// TIA Portal project "LinkedList_v000_000_008" (V16)
// task for 000.000.007: create LinkedList.Insert

(* hardware
DEVICE "S7-1200 station_1"  S7-1200 Station
   slot 0: "Rack_0"  S7-1200 Rack  Rack  V1.0
   slot 1: "PLC_1"  CPU 1212C DC/DC/DC  6ES7 212-1AE40-0XB0  V4.4
*)

// ===== PLC "PLC_1"  CPU 1212C DC/DC/DC =====

VAR_GLOBAL   // PLC tag table "Default tag table"
   "System_Byte" AT %MB1 : Byte;
   "FirstScan" AT %M1.0 : Bool;
   "DiagStatusUpdate" AT %M1.1 : Bool;
   "AlwaysTRUE" AT %M1.2 : Bool;
   "AlwaysFALSE" AT %M1.3 : Bool;
   "Clock_Byte" AT %MB0 : Byte;
   "Clock_10Hz" AT %M0.0 : Bool;
   "Clock_5Hz" AT %M0.1 : Bool;
   "Clock_2.5Hz" AT %M0.2 : Bool;
   "Clock_2Hz" AT %M0.3 : Bool;
   "Clock_1.25Hz" AT %M0.4 : Bool;
   "Clock_1Hz" AT %M0.5 : Bool;
   "Clock_0.625Hz" AT %M0.6 : Bool;
   "Clock_0.5Hz" AT %M0.7 : Bool;
END_VAR

VAR_GLOBAL CONSTANT   // PLC tag table "Default tag table"
   "NULL_TOKEN" : DInt := -1;
   "AVAILABLE_SLOT" : DInt := -1;
   "TAIL_ADDRESS" : DInt := -2;
   "NOT_FOUND_FLAG" : DInt := -1;
END_VAR

TYPE "LinkedList.Node.Payload.UDT"
   STRUCT
      id : Char;
      status : String;
   END_STRUCT;
END_TYPE

TYPE "LinkedList.Node.UDT"
   STRUCT
      payload : "LinkedList.Node.Payload.UDT";
      pointer : DInt := -1;
   END_STRUCT;
END_TYPE

TYPE "LinkedList.UDT"
   STRUCT
      head : DInt := -1;
      list : Array[0..4] of "LinkedList.Node.UDT";
   END_STRUCT;
END_TYPE

TYPE "Validate.LinkedList.FindPointer.UDT"
   STRUCT
      request : Bool;
      needle : DInt;
      not_found : DInt;
      index : DInt;
   END_STRUCT;
END_TYPE

TYPE "Validate.LinkedList.FindPayload.UDT"
   STRUCT
      request : Bool;
      needle : "LinkedList.Node.Payload.UDT";
      not_found : DInt;
      tail_address : DInt;
      index : DInt;
   END_STRUCT;
END_TYPE

TYPE "Validate.LinkedList.FindID.UDT"
   STRUCT
      request : Bool;
      needle : Char;
      not_found : DInt;
      tail_address : DInt;
      index : DInt;
   END_STRUCT;
END_TYPE

TYPE "Validate.LinkedList.FindStatus.UDT"
   STRUCT
      request : Bool;
      needle : String;
      not_found : DInt;
      tail_address : DInt;
      index : DInt;
   END_STRUCT;
END_TYPE

TYPE "Validate.LinkedList.AddHead.UDT"
   STRUCT
      request : Bool;
      available_slot : DInt := -1;
      payload : "LinkedList.Node.Payload.UDT";
      tail_address : DInt := -2;
      status : String;
   END_STRUCT;
END_TYPE

TYPE "Validate.LinkedList.RemoveHead.UDT"
   STRUCT
      request : Bool;
      status : String;
   END_STRUCT;
END_TYPE

TYPE "Validate.LinkedList.FindPrevious.UDT"
   STRUCT
      request : Bool;
      needle : "LinkedList.Node.Payload.UDT";
      not_found : DInt;
      tail_address : DInt;
      index : DInt;
   END_STRUCT;
END_TYPE

TYPE "Validate.LinkedList.RemoveNode.UDT"
   STRUCT
      request : Bool;
      payload : "LinkedList.Node.Payload.UDT";
      null_token : DInt := -1;
      tail_address : DInt := -2;
      status : String;
   END_STRUCT;
END_TYPE

TYPE "Validate.LinkedList.Append.UDT"
   STRUCT
      request : Bool;
      payload : "LinkedList.Node.Payload.UDT";
      available_slot : DInt := -1;
      tail_address : DInt := -2;
      status : String;
   END_STRUCT;
END_TYPE

TYPE "Validate.LinkedList.Insert.UDT"
   STRUCT
      request : Bool;
      payload : "LinkedList.Node.Payload.UDT";
      after : "LinkedList.Node.Payload.UDT";
      available_slot : DInt := -1;
      not_found : DInt := -1;
      tail_address : DInt := -2;
      status : String;
   END_STRUCT;
END_TYPE

TYPE "Validate.LinkedList.Clear.UDT"
   STRUCT
      request : Bool;
      available_slot : DInt := -1;
      tail_address : DInt := -2;
      status : String;
   END_STRUCT;
END_TYPE

TYPE "Validate.LinkedList.AddNode.UDT"
   STRUCT
      request : Bool;
      available_slot : DInt := -1;
      payload : "LinkedList.Node.Payload.UDT";
      tail_address : DInt := -2;
      status : String;
   END_STRUCT;
END_TYPE

DATA_BLOCK "LinkedList.IDB"   // DB1
{ S7_Optimized_Access := 'TRUE' }
AUTHOR : Machado
FAMILY : LinkedList
VERSION : 0.1
// stored: InstanceOfName LinkedList
"LinkedList"
BEGIN
END_DATA_BLOCK

DATA_BLOCK "ValidationSignals"   // DB2
{ S7_Optimized_Access := 'TRUE' }
VERSION : 0.1
   VAR
      FindPointer : "Validate.LinkedList.FindPointer.UDT";
      FindPayload : "Validate.LinkedList.FindPayload.UDT";
      FindID : "Validate.LinkedList.FindID.UDT";
      FindStatus : "Validate.LinkedList.FindStatus.UDT";
      AddHead : "Validate.LinkedList.AddHead.UDT";
      RemoveHead : "Validate.LinkedList.RemoveHead.UDT";
      FindPrevious : "Validate.LinkedList.FindPrevious.UDT";
      RemoveNode : "Validate.LinkedList.RemoveNode.UDT";
      AppendNode : "Validate.LinkedList.Append.UDT";
      InsertNode : "Validate.LinkedList.Insert.UDT";
      Clear : "Validate.LinkedList.Clear.UDT";
      AddNode : "Validate.LinkedList.AddNode.UDT";
   END_VAR
BEGIN
END_DATA_BLOCK

FUNCTION_BLOCK "LinkedList"   // FB1, SCL
TITLE = Linked List
{ S7_Optimized_Access := 'TRUE' }
AUTHOR : Machado
FAMILY : LinkedList
VERSION : 0.1
   VAR_INPUT
      request : DInt;
   END_VAR
   VAR
      list : "LinkedList.UDT";
      requests : "LinkedList.UDT";
   END_VAR
   VAR_TEMP
      test : DInt;
   END_VAR
BEGIN
   CASE #request OF
       0:  // Statement section case 1
           ;
       2..4:  // Statement section case 2 to 4
           ;
       ELSE  // Statement section ELSE
           ;
   END_CASE;
END_FUNCTION_BLOCK

FUNCTION "LinkedList.FindPointer" : DInt   // FC1, SCL
TITLE = Find Node by Pointer In Linked List
{ S7_Optimized_Access := 'TRUE' }
AUTHOR : Machado
FAMILY : LinkedList
VERSION : 0.1
// returns not_found when not found.
// otherwise returs index of parent array where node with needle value as pointer.
   VAR_INPUT
      needle : DInt;
      not_found : DInt;   // value returned to user if needle not found
   END_VAR
   VAR_IN_OUT
      haystack : "LinkedList.UDT";
   END_VAR
   VAR_TEMP
      i : DInt;
      size : DInt;
   END_VAR
BEGIN
   REGION "GET SIZE"
       #size := UDINT_TO_DINT("LinkedList.Node[].CountOfElements"(#haystack.list));
   END_REGION


   REGION "SEARCH"
       FOR #i := 0 TO #size - 1 DO
           // no match
           IF #haystack.list[#i]."pointer" <> #needle THEN
               CONTINUE;
           END_IF;
           // match
           #"LinkedList.FindPointer" := #i;
           RETURN;
       END_FOR;
   END_REGION


   REGION "NOT FOUND"
       #"LinkedList.FindPointer" := #not_found;
       RETURN;
   END_REGION
END_FUNCTION

FUNCTION "LinkedList.Node[].CountOfElements" : UDInt   // FC2, SCL
TITLE = Count Of Elements of an Array of Linked List Nodes
{ S7_Optimized_Access := 'TRUE' }
AUTHOR : Machado
FAMILY : LinkedList
VERSION : 0.1
   VAR_INPUT
      list : Variant;
   END_VAR
BEGIN
   #"LinkedList.Node[].CountOfElements" := CountOfElements(#list);
   RETURN;
END_FUNCTION

FUNCTION "LinkedList.FindPayload" : DInt   // FC3, SCL
TITLE = Finde Node Index By Payload
{ S7_Optimized_Access := 'TRUE' }
AUTHOR : Machado
FAMILY : LinkedList
VERSION : 0.1
   VAR_INPUT
      needle : "LinkedList.Node.Payload.UDT";
      not_found : DInt;
      tail_address : DInt;
   END_VAR
   VAR_IN_OUT
      haystack : "LinkedList.UDT";
   END_VAR
   VAR_TEMP
      size : DInt;
      this_node : "LinkedList.Node.UDT";
      next_node : "LinkedList.Node.UDT";
      nodes_visited : DInt;
   END_VAR
BEGIN
   REGION "GET SIZE"
       #size := UDINT_TO_DINT("LinkedList.Node[].CountOfElements"(#haystack.list));
   END_REGION


   REGION "PRE-CONDITIONS"
       IF NOT "DInt.InRange"(x := #haystack.head, max := #size - 1, min := 0) THEN
           #"LinkedList.FindPayload" := #not_found;
           RETURN;
       END_IF;
   END_REGION


   REGION "PRIME WHILE LOOP"
       #this_node := #haystack.list[#haystack.head];
       IF #this_node.payload = #needle THEN
           #"LinkedList.FindPayload" := #haystack.head;
           RETURN;
       END_IF;
       #nodes_visited := 1;
   END_REGION


   REGION "SEARCH"
       WHILE #this_node."pointer" <> #tail_address DO
           #next_node := #haystack.list[#this_node."pointer"];
           IF #next_node.payload = #needle THEN
               #"LinkedList.FindPayload" := #this_node."pointer";
               RETURN;
           END_IF;
           #nodes_visited += 1;
           IF #nodes_visited > #size THEN
               #"LinkedList.FindPayload" := #not_found;
               RETURN;
           END_IF;
           #this_node := #next_node;
       END_WHILE;
   END_REGION


   REGION "NOT FOUND"
       #"LinkedList.FindPayload" := #not_found;
       RETURN;
   END_REGION
END_FUNCTION

FUNCTION "DInt.InRange" : Bool   // FC4, SCL
TITLE = Value Is In Range
{ S7_Optimized_Access := 'TRUE' }
AUTHOR : Machado
FAMILY : DInt
VERSION : 0.1
   VAR_INPUT
      x : DInt;
      max : DInt;
      min : DInt;
   END_VAR
BEGIN
   #"DInt.InRange" := #min <= #x AND #x <= #max;
END_FUNCTION

FUNCTION "LinkedList.FindID" : DInt   // FC5, SCL
TITLE = Finde Node Index By Payload
{ S7_Optimized_Access := 'TRUE' }
AUTHOR : Machado
FAMILY : LinkedList
VERSION : 0.1
   VAR_INPUT
      needle : Char;
      not_found : DInt;
      tail_address : DInt;
   END_VAR
   VAR_IN_OUT
      haystack : "LinkedList.UDT";
   END_VAR
   VAR_TEMP
      size : DInt;
      this_node : "LinkedList.Node.UDT";
      next_node : "LinkedList.Node.UDT";
      nodes_visited : DInt;
   END_VAR
BEGIN
   REGION "GET SIZE"
       #size := UDINT_TO_DINT("LinkedList.Node[].CountOfElements"(#haystack.list));
   END_REGION


   REGION "PRE-CONDITIONS"
       IF NOT "DInt.InRange"(x := #haystack.head, max := #size - 1, min := 0) THEN
           #"LinkedList.FindID" := #not_found;
           RETURN;
       END_IF;
   END_REGION


   REGION "PRIME WHILE LOOP"
       #this_node := #haystack.list[#haystack.head];
       IF #this_node.payload.id = #needle THEN
           #"LinkedList.FindID" := #haystack.head;
           RETURN;
       END_IF;
       #nodes_visited := 1;
   END_REGION


   REGION "SEARCH"
       WHILE #this_node."pointer" <> #tail_address DO
           #next_node := #haystack.list[#this_node."pointer"];
           IF #next_node.payload.id = #needle THEN
               #"LinkedList.FindID" := #this_node."pointer";
               RETURN;
           END_IF;
           #nodes_visited += 1;
           IF #nodes_visited > #size THEN
               #"LinkedList.FindID" := #not_found;
               RETURN;
           END_IF;
           #this_node := #next_node;
       END_WHILE;
   END_REGION


   REGION "NOT FOUND"
       #"LinkedList.FindID" := #not_found;
       RETURN;
   END_REGION
END_FUNCTION

FUNCTION "LinkedList.FindStatus" : DInt   // FC6, SCL
TITLE = Finde Node Index By Payload
{ S7_Optimized_Access := 'TRUE' }
AUTHOR : Machado
FAMILY : LinkedList
VERSION : 0.1
   VAR_INPUT
      needle : String;
      not_found : DInt;
      tail_address : DInt;
   END_VAR
   VAR_IN_OUT
      haystack : "LinkedList.UDT";
   END_VAR
   VAR_TEMP
      size : DInt;
      this_node : "LinkedList.Node.UDT";
      next_node : "LinkedList.Node.UDT";
      nodes_visited : DInt;
   END_VAR
BEGIN
   REGION "GET SIZE"
       #size := UDINT_TO_DINT("LinkedList.Node[].CountOfElements"(#haystack.list));
   END_REGION


   REGION "PRE-CONDITIONS"
       IF NOT "DInt.InRange"(x := #haystack.head, max := #size - 1, min := 0) THEN
           #"LinkedList.FindStatus" := #not_found;
           RETURN;
       END_IF;
   END_REGION


   REGION "PRIME WHILE LOOP"
       #this_node := #haystack.list[#haystack.head];
       IF #this_node.payload.status = #needle THEN
           #"LinkedList.FindStatus" := #haystack.head;
           RETURN;
       END_IF;
       #nodes_visited := 1;
   END_REGION


   REGION "SEARCH"
       WHILE #this_node."pointer" <> #tail_address DO
           #next_node := #haystack.list[#this_node."pointer"];
           IF #next_node.payload.status = #needle THEN
               #"LinkedList.FindStatus" := #this_node."pointer";
               RETURN;
           END_IF;
           #nodes_visited += 1;
           IF #nodes_visited > #size THEN
               #"LinkedList.FindStatus" := #not_found;
               RETURN;
           END_IF;
           #this_node := #next_node;
       END_WHILE;
   END_REGION


   REGION "NOT FOUND"
       #"LinkedList.FindStatus" := #not_found;
       RETURN;
   END_REGION
END_FUNCTION

FUNCTION "LinkedList.AddHead" : String   // FC7, SCL
TITLE = Add a Head Node to a Linked List
{ S7_Optimized_Access := 'TRUE' }
AUTHOR : Machado
FAMILY : LinkedList
VERSION : 0.1
// Use this in your linked list. Instantiates LinkedList.CreateHead and LinkedList.ReplaceHead when appropriate.
   VAR_INPUT
      available_slot : DInt;
      payload : "LinkedList.Node.Payload.UDT";
      tail_address : DInt;
   END_VAR
   VAR_IN_OUT
      list : "LinkedList.UDT";
   END_VAR
   VAR_TEMP
      message : String;
   END_VAR
BEGIN
   REGION "NO HEAD"
       IF #list.head = -1 THEN
           #message := "LinkedList.CreateHead"(available_slot := #available_slot,
                                               payload := #payload,
                                               tail_address := #tail_address,
                                               list := #list);
           #"LinkedList.AddHead" := #message;
           RETURN;
       END_IF;
   END_REGION
   REGION "REPLACE HEAD"
       #message := "LinkedList.ReplaceHead"(available_slot := #available_slot,
                                            payload := #payload,
                                            tail_address := #tail_address,
                                            list := #list);
       #"LinkedList.AddHead" := #message;
       RETURN;
   END_REGION
END_FUNCTION

FUNCTION "LinkedList.CreateHead" : String   // FC8, SCL
TITLE = Create a New Head Node for a Linked List
{ S7_Optimized_Access := 'TRUE' }
AUTHOR : Machado
FAMILY : LinkedList
VERSION : 0.1
   VAR_INPUT
      available_slot : DInt;
      payload : "LinkedList.Node.Payload.UDT";
      tail_address : DInt;
   END_VAR
   VAR_IN_OUT
      list : "LinkedList.UDT";
   END_VAR
   VAR_TEMP
      first_available_slot : DInt;
      message : String;
   END_VAR
   VAR CONSTANT
      CREATED : String := 'head created';
      FULL : String := 'no space in array. head not created.';
      NOT_FOUND : DInt := -1;
   END_VAR
BEGIN
   REGION "GET FIRST AVAILABLE SLOT"
       #first_available_slot := "LinkedList.FindPointer"(needle := #available_slot,
                                                         not_found := #NOT_FOUND,
                                                         haystack := #list);
   END_REGION


   REGION "NO ROOM IN LIST"
       IF #first_available_slot = #NOT_FOUND THEN
           #"LinkedList.CreateHead" := #FULL;
           RETURN;
       END_IF;
   END_REGION


   REGION "CREATE HEAD"
       #message := "LinkedList.Clear"(available_slot := #available_slot,
                                      tail_address := #tail_address,
                                      list := #list);
       #list.head := #first_available_slot;
       #list.list[#first_available_slot].payload := #payload;
       #list.list[#first_available_slot]."pointer" := #tail_address;
       #"LinkedList.CreateHead" := #CREATED;
       RETURN;
   END_REGION
END_FUNCTION

FUNCTION "LinkedList.ReplaceHead" : String   // FC9, SCL
TITLE = Replace Linked List's Existing Head Node
{ S7_Optimized_Access := 'TRUE' }
AUTHOR : Machado
FAMILY : LinkedList
VERSION : 0.1
   VAR_INPUT
      available_slot : DInt;
      payload : "LinkedList.Node.Payload.UDT";
      tail_address : DInt;
   END_VAR
   VAR_IN_OUT
      list : "LinkedList.UDT";
   END_VAR
   VAR_TEMP
      first_available_slot : DInt;
   END_VAR
   VAR CONSTANT
      FULL : String := 'no space in array. new head not added.';
      ADDED : String := 'new head added';
      NOT_FOUND : DInt := -1;
   END_VAR
BEGIN
   REGION "GET FIRST AVAILABLE SLOT"
       #first_available_slot := "LinkedList.FindPointer"(needle := #available_slot,
                                                         not_found := #NOT_FOUND,
                                                         haystack := #list);
   END_REGION


   REGION "NO ROOM IN LIST"
       IF #first_available_slot = #NOT_FOUND THEN
           #"LinkedList.ReplaceHead" := #FULL;
           RETURN;
       END_IF;
   END_REGION


   REGION "CREATE HEAD"
       #list.list[#first_available_slot].payload := #payload;
       #list.list[#first_available_slot]."pointer" := #list.head;
       #list.head := #first_available_slot;
       #"LinkedList.ReplaceHead" := #ADDED;
       RETURN;
   END_REGION
END_FUNCTION

FUNCTION "LinkedList.DeleteNode" : "LinkedList.Node.UDT"   // FC10, SCL
TITLE = Delete a Node from a Linked List
{ S7_Optimized_Access := 'TRUE' }
AUTHOR : Machado
FAMILY : LinkedList
VERSION : 0.1
   VAR_INPUT
      null_token : DInt;
   END_VAR
   VAR_TEMP
      node : "LinkedList.Node.UDT";
   END_VAR
BEGIN
   #node."pointer" := #null_token;
   #"LinkedList.DeleteNode" := #node;
   RETURN;
END_FUNCTION

FUNCTION "LinkedList.RemoveHead" : String   // FC11, SCL
TITLE = Remove Head Node from a Linked List
{ S7_Optimized_Access := 'TRUE' }
AUTHOR : Machado
FAMILY : LinkedList
VERSION : 0.1
// no head: returns no head message
// has head: removes, returns removed head message
   VAR_INPUT
      null_token : DInt;
   END_VAR
   VAR_IN_OUT
      list : "LinkedList.UDT";
   END_VAR
   VAR_TEMP
      head_pointer : DInt;
   END_VAR
   VAR CONSTANT
      NO_HEAD : String := 'no head, no operation';
      HEAD_REMOVED : String := 'head removed';
      HEAD_INDEX_OUT_OF_BOUNDS : String := 'head index out of bounds. no operation.';
   END_VAR
BEGIN
   REGION "NO HEAD"
       IF #list.head < 0 THEN
           #"LinkedList.RemoveHead" := #NO_HEAD;
           RETURN;
       END_IF;
   END_REGION


   REGION "HEAD POINTER IS OUT OF BOUNDS"
       IF #list.head >= UDINT_TO_DINT("LinkedList.Node[].CountOfElements"(#list.list))THEN
           #"LinkedList.RemoveHead" := #HEAD_INDEX_OUT_OF_BOUNDS;
           RETURN;
       END_IF;
   END_REGION


   REGION "HAS HEAD"
       #head_pointer := #list.list[#list.head]."pointer";
       #list.list[#list.head] := "LinkedList.DeleteNode"(#null_token);
       #list.head := #head_pointer;
       #"LinkedList.RemoveHead" := #HEAD_REMOVED;
       RETURN;
   END_REGION
END_FUNCTION

FUNCTION "LinkedList.FindPrevious" : DInt   // FC12, SCL
TITLE = Finde Node Index By Payload
{ S7_Optimized_Access := 'TRUE' }
AUTHOR : Machado
FAMILY : LinkedList
VERSION : 0.1
   VAR_INPUT
      needle : "LinkedList.Node.Payload.UDT";
      not_found : DInt;
      tail_address : DInt;
   END_VAR
   VAR_IN_OUT
      haystack : "LinkedList.UDT";
   END_VAR
   VAR_TEMP
      size : DInt;
      this_node : "LinkedList.Node.UDT";
      this_node_index : DInt;
      next_node : "LinkedList.Node.UDT";
      nodes_visited : DInt;
   END_VAR
BEGIN
   REGION "GET SIZE"
       #size := UDINT_TO_DINT("LinkedList.Node[].CountOfElements"(#haystack.list));
   END_REGION


   REGION "PRE-CONDITIONS"
       IF NOT "DInt.InRange"(x := #haystack.head, max := #size - 1, min := 0) THEN
           #"LinkedList.FindPrevious" := #not_found;
           RETURN;
       END_IF;
   END_REGION


   REGION "PRIME WHILE LOOP"
       #this_node_index := #haystack.head;
       #this_node := #haystack.list[#haystack.head];
       IF #this_node.payload = #needle THEN
           #"LinkedList.FindPrevious" := #not_found;
           RETURN;
       END_IF;
       #nodes_visited := 1;
   END_REGION


   REGION "SEARCH"
       WHILE #this_node."pointer" <> #tail_address DO
           #next_node := #haystack.list[#this_node."pointer"];
           IF #next_node.payload = #needle THEN
               #"LinkedList.FindPrevious" := #this_node_index;
               RETURN;
           END_IF;
           #nodes_visited += 1;
           IF #nodes_visited >= #size THEN
               #"LinkedList.FindPrevious" := #not_found;
               RETURN;
           END_IF;
           #this_node_index := #this_node."pointer";
           #this_node := #next_node;
       END_WHILE;
   END_REGION


   REGION "NOT FOUND"
       #"LinkedList.FindPrevious" := #not_found;
       RETURN;
   END_REGION
END_FUNCTION

FUNCTION "LinkedList.RemoveNode" : String   // FC13, SCL
TITLE = Removes a Node From a Linked List
{ S7_Optimized_Access := 'TRUE' }
AUTHOR : Machado
FAMILY : LinkedList
VERSION : 0.1
   VAR_INPUT
      node_payload : "LinkedList.Node.Payload.UDT";
      null_token : DInt;
      tail_address : DInt;
   END_VAR
   VAR_IN_OUT
      list : "LinkedList.UDT";
   END_VAR
   VAR_TEMP
      previous_node_index : DInt;
      this_node_index : DInt;
      list_size : DInt;
   END_VAR
   VAR CONSTANT
      EMPTY_LIST : String := 'list empty. no operation.';
      NOT_FOUND : String := 'payload not found. no operation.';
      INVALID_INDEX : String := 'node found but at invalid array index. no operation.';
      SUCCESS : String := 'node removed from list.';
   END_VAR
BEGIN
   REGION "LIST IS EMPTY"
       IF #list.head < 0 THEN
           #"LinkedList.RemoveNode" := #EMPTY_LIST;
           RETURN;
       END_IF;
   END_REGION


   REGION "GET PREVIOUS NODE INDEX"
       #previous_node_index := "LinkedList.FindPrevious"(needle := #node_payload,
                                                         not_found := #null_token,
                                                         tail_address := #tail_address,
                                                         haystack := #list);
   END_REGION


   REGION "NODE NOT FOUND"
       IF #previous_node_index = #null_token THEN
           #"LinkedList.RemoveNode" := #NOT_FOUND;
           RETURN;
       END_IF;
   END_REGION


   REGION "GET THIS NODE INDEX"
       #this_node_index := #list.list[#previous_node_index]."pointer";
   END_REGION


   REGION "FOUND NODE INDEX INVALID"
       #list_size := UDINT_TO_DINT("LinkedList.Node[].CountOfElements"(#list.list));
       IF NOT "DInt.InRange"(x := #previous_node_index, max := #list_size - 1, min := 0) THEN
           #"LinkedList.RemoveNode" := #INVALID_INDEX;
           RETURN;
       END_IF;
       IF NOT "DInt.InRange"(x := #this_node_index, max := #list_size - 1, min := 0) THEN
           #"LinkedList.RemoveNode" := #INVALID_INDEX;
           RETURN;
       END_IF;
   END_REGION


   REGION "REMOVE"
       #list.list[#previous_node_index]."pointer" := #list.list[#this_node_index]."pointer";
       #list.list[#this_node_index] := "LinkedList.DeleteNode"(#null_token);
       #"LinkedList.RemoveNode" := #SUCCESS;
       RETURN;
   END_REGION
END_FUNCTION

FUNCTION "LinkedList.AppendNode" : String   // FC14, SCL
TITLE = Append New Node to End of Linked List
{ S7_Optimized_Access := 'TRUE' }
AUTHOR : Machado
FAMILY : LinkedList
VERSION : 0.1
   VAR_INPUT
      available_slot : DInt;
      payload : "LinkedList.Node.Payload.UDT";
      tail_address : DInt;
   END_VAR
   VAR_IN_OUT
      list : "LinkedList.UDT";
   END_VAR
   VAR_TEMP
      first_slot : DInt;
      size : DInt;
      tail : DInt;
   END_VAR
   VAR CONSTANT
      NOT_FOUND : DInt := -1;
      NO_AVAILABLE_SLOT : String := 'no available slot. no operation.';
      TAIL_NOT_FOUND : String := 'tail node not found. no operation.';
      TAIL_INDEX_NOT_IN_RANGE : String := 'tail index not in range. no operation';
      NODE_APPENDED : String := 'node appended';
   END_VAR
BEGIN
   REGION "GET FIRST SLOT"
       #first_slot := "LinkedList.FindPointer"(needle := #available_slot,
                                               not_found := #NOT_FOUND,
                                               haystack := #list);
   END_REGION


   REGION "NO SLOT AVAILABLE"
       IF #first_slot = #NOT_FOUND THEN
           #"LinkedList.AppendNode" := #NO_AVAILABLE_SLOT;
           RETURN;
       END_IF;
   END_REGION


   REGION "GET TAIL INDEX"
       #tail := "LinkedList.FindPointer"(needle := #tail_address,
                                         not_found := #NOT_FOUND,
                                         haystack := #list);
   END_REGION


   REGION "TAIL NOT FOUND"
       IF #tail = #NOT_FOUND THEN
           #"LinkedList.AppendNode" := #TAIL_NOT_FOUND;
           RETURN;
       END_IF;
   END_REGION


   REGION "TAIL INDEX NOT IN RANGE"
       #size := UDINT_TO_DINT("LinkedList.Node[].CountOfElements"(#list.list));
       IF NOT "DInt.InRange"(x := #tail, max := #size - 1, min := 0) THEN
           #"LinkedList.AppendNode" := #TAIL_INDEX_NOT_IN_RANGE;
           RETURN;
       END_IF;
   END_REGION


   REGION "APPEND"
       #list.list[#tail]."pointer" := #first_slot;
       #list.list[#first_slot].payload := #payload;
       #list.list[#first_slot]."pointer" := #tail_address;
       #"LinkedList.AppendNode" := #NODE_APPENDED;
       RETURN;
   END_REGION
END_FUNCTION

FUNCTION "LinkedList.InsertNode" : String   // FC15, SCL
TITLE = Insert a New Node into a Linked List
{ S7_Optimized_Access := 'TRUE' }
AUTHOR : Machado
FAMILY : LinkedList
VERSION : 0.1
   VAR_INPUT
      payload : "LinkedList.Node.Payload.UDT";
      after : "LinkedList.Node.Payload.UDT";
      available_slot : DInt;
      tail_address : DInt;
   END_VAR
   VAR_IN_OUT
      list : "LinkedList.UDT";
   END_VAR
   VAR_TEMP
      after_index : DInt;
      available_index : DInt;
      message : String;
      size : DInt;
   END_VAR
   VAR CONSTANT
      NOT_FOUND : DInt := -1;
      NO_AVAILABLE_SLOT : String := 'no available slot in parent array. no operation.';
      AFTER_NOT_FOUND : String := '"after" node not found. no operation.';
      NODE_INSERTED : String := 'node inserted.';
      AFTER_INDEX_INVALID : String := '"after" node index invalid. no operation.';
   END_VAR
BEGIN
   REGION "SLOT NOT AVAILABLE"
       #available_index := "LinkedList.FindPointer"(needle := #available_slot,
                                               not_found := #NOT_FOUND,
                                               haystack := #list);
       IF #available_index = #NOT_FOUND THEN
           #"LinkedList.InsertNode" := #NO_AVAILABLE_SLOT;
           RETURN;
       END_IF;
   END_REGION


   REGION "AFTER NODE NOT FOUND"
       #after_index := "LinkedList.FindPayload"(needle := #after,
                                                not_found := #NOT_FOUND,
                                                tail_address := #tail_address,
                                                haystack := #list);
       IF #after_index = #NOT_FOUND THEN
           #"LinkedList.InsertNode" := #AFTER_NOT_FOUND;
           RETURN;
       END_IF;
   END_REGION


   REGION "AFTER INDEX INVALID"
       #size := UDINT_TO_DINT("LinkedList.Node[].CountOfElements"(#list.list));
       IF NOT "DInt.InRange"(x:=#after_index, max:=#size-1, min:=0) THEN
           #"LinkedList.InsertNode" := #AFTER_INDEX_INVALID;
           RETURN;
       END_IF;
   END_REGION


   REGION "AFTER IS TAIL"
       IF #list.list[#after_index]."pointer" = #tail_address THEN
           #message := "LinkedList.AppendNode"(payload := #payload,
                                               available_slot := #available_slot,
                                               tail_address := #tail_address,
                                               list := #list);
           #"LinkedList.InsertNode" := #message;
           RETURN;
       END_IF;
   END_REGION


   REGION "INSERT"
       #list.list[#available_index].payload := #payload;
       #list.list[#available_index]."pointer" := #list.list[#after_index]."pointer";
       #list.list[#after_index]."pointer" := #available_index;
       #"LinkedList.InsertNode" := #NODE_INSERTED;
       RETURN;
   END_REGION
END_FUNCTION

FUNCTION "LinkedList.Clear" : String   // FC16, SCL
TITLE = Clear a Linked List of All Nodes
{ S7_Optimized_Access := 'TRUE' }
AUTHOR : Machado
FAMILY : LinkedList
VERSION : 0.1
   VAR_INPUT
      available_slot : DInt;
      tail_address : DInt;
   END_VAR
   VAR_IN_OUT
      list : "LinkedList.UDT";
   END_VAR
   VAR_TEMP
      i : DInt;
      size : DInt;
      this_node_index : DInt;
      next_node_index : DInt;
   END_VAR
   VAR CONSTANT
      COMPLETE : String := 'list cleared of all nodes.';
   END_VAR
BEGIN
   REGION "CLEAR"
       #size := UDINT_TO_DINT("LinkedList.Node[].CountOfElements"(#list.list));
       FOR #i := 0 TO #size - 1 DO
           #list.list[#i] := "LinkedList.DeleteNode"(#available_slot);
       END_FOR;
   END_REGION 


   (*
   REGION "PRIME WHILE"
       #next_node_index := #list.list[#list.head]."pointer";
       #list.list[#list.head] := "LinkedList.DeleteNode"(#available_slot);
       #this_node_index := #next_node_index;
   END_REGION

   REGION "CLEAR"
       WHILE #this_node_index <> #tail_address AND #this_node_index <> #available_slot DO
           #next_node_index := #list.list[#this_node_index]."pointer";
           #list.list[#this_node_index] := "LinkedList.DeleteNode"(#available_slot);
           #this_node_index := #next_node_index;
       END_WHILE;
   END_REGION
   *)


   REGION "RETURN"
       #list.head := #tail_address;
       #"LinkedList.Clear" := #COMPLETE;
       RETURN;
   END_REGION
END_FUNCTION

FUNCTION "LinkedList.AddNode" : String   // FC17, SCL
TITLE = Add a Node to a Linked list
{ S7_Optimized_Access := 'TRUE' }
AUTHOR : Machado
FAMILY : LinkedList
VERSION : 0.1
// adds a node as either a head (if a blank list) or a new tail (if a populated list).
   VAR_INPUT
      available_slot : DInt;
      payload : "LinkedList.Node.Payload.UDT";
      tail_address : DInt;
   END_VAR
   VAR_IN_OUT
      list : "LinkedList.UDT";
   END_VAR
   VAR_TEMP
      first_slot : DInt;
      message : String;
      size : DInt;
   END_VAR
   VAR CONSTANT
      NOT_FOUND : DInt := -1;
      ARRAY_FULL : String := 'parent array full. no operation.';
   END_VAR
BEGIN
   REGION "GET FIRST AVAILABLE"
       #first_slot := "LinkedList.FindPointer"(needle := #available_slot,
                                               not_found := #NOT_FOUND,
                                               haystack := #list);
   END_REGION


   REGION "LIST FULL"
       IF #first_slot = #NOT_FOUND THEN
           #"LinkedList.AddNode" := #ARRAY_FULL;
           RETURN;
       END_IF;
   END_REGION


   REGION "LIST HEAD INDEX INVALID"
       #size := UDINT_TO_DINT("LinkedList.Node[].CountOfElements"(#list.list));
       IF NOT "DInt.InRange"(x:=#list.head, max:=#size-1, min:=0) THEN
           #message := "LinkedList.CreateHead"(available_slot := #available_slot,
                                               payload := #payload,
                                               tail_address := #tail_address,
                                               list := #list);
           #"LinkedList.AddNode" := #message;
           RETURN;
       END_IF;
   END_REGION


   REGION "LIST EMPTY"
       IF #list.head = #tail_address THEN
           #message := "LinkedList.CreateHead"(available_slot := #available_slot,
                                               payload := #payload,
                                               tail_address := #tail_address,
                                               list := #list);
           #"LinkedList.AddNode" := #message;
           RETURN;
       END_IF;
   END_REGION


   REGION "APPEND"
       #message := "LinkedList.AppendNode"(available_slot := #available_slot,
                                           payload := #payload,
                                           tail_address := #tail_address,
                                           list := #list);
       #"LinkedList.AddNode" := #message;
       RETURN;
   END_REGION
END_FUNCTION

ORGANIZATION_BLOCK "Main"   // OB1, LAD, ProgramCycle
TITLE = "Main Program Sweep (Cycle)"
{ S7_Optimized_Access := 'TRUE' }
VERSION : 0.1
   VAR_INPUT
      Initial_Call : Bool;   // Initial call of this OB
      Remanence : Bool;   // =True, if remanent data are available
   END_VAR
   VAR_TEMP   // added for the SCL form of the ladder/FBD networks
      _w1 : Bool;
   END_VAR
BEGIN

REGION Network 1: CALL LINKED LIST
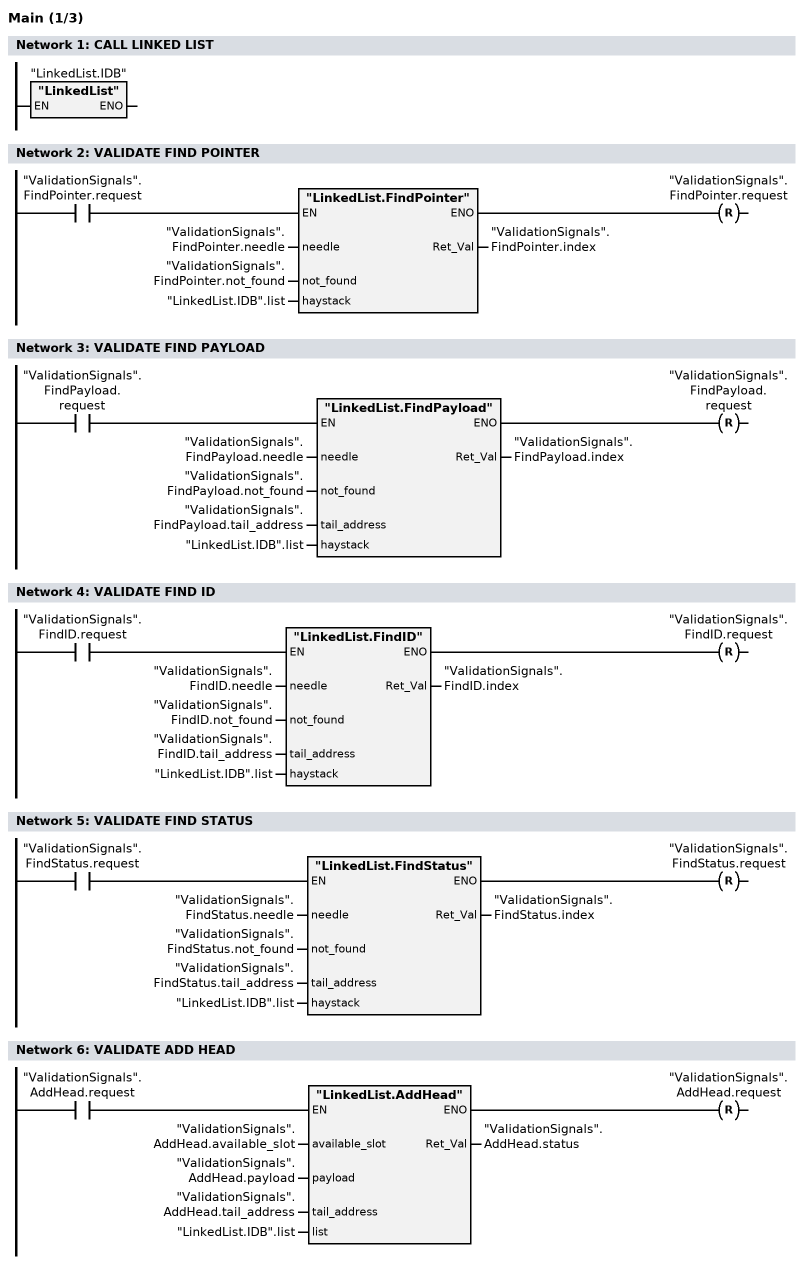
   RUNG wire#powerrail
      "LinkedList.IDB"()
   END_RUNG
   // the same network as SCL:
   "LinkedList.IDB"();   // "LinkedList"
END_REGION

REGION Network 2: VALIDATE FIND POINTER
   RUNG wire#powerrail
      Contact( "ValidationSignals".FindPointer.request )
      "LinkedList.FindPointer"(needle := "ValidationSignals".FindPointer.needle, not_found := "ValidationSignals".FindPointer.not_found, haystack := "LinkedList.IDB".list, Ret_Val => "ValidationSignals".FindPointer.index)
      R_Coil( "ValidationSignals".FindPointer.request )
   END_RUNG
   // the same network as SCL:
   "ValidationSignals".FindPointer.index := "LinkedList.FindPointer"(EN := "ValidationSignals".FindPointer.request,
                           needle := "ValidationSignals".FindPointer.needle,
                           not_found := "ValidationSignals".FindPointer.not_found,
                           haystack := "LinkedList.IDB".list,
                           ENO => #_w1);
   IF #_w1 THEN "ValidationSignals".FindPointer.request := FALSE; END_IF;
END_REGION

REGION Network 3: VALIDATE FIND PAYLOAD
   RUNG wire#powerrail
      Contact( "ValidationSignals".FindPayload.request )
      "LinkedList.FindPayload"(needle := "ValidationSignals".FindPayload.needle, not_found := "ValidationSignals".FindPayload.not_found, tail_address := "ValidationSignals".FindPayload.tail_address, haystack := "LinkedList.IDB".list, Ret_Val => "ValidationSignals".FindPayload.index)
      R_Coil( "ValidationSignals".FindPayload.request )
   END_RUNG
   // the same network as SCL:
   "ValidationSignals".FindPayload.index := "LinkedList.FindPayload"(EN := "ValidationSignals".FindPayload.request,
                           needle := "ValidationSignals".FindPayload.needle,
                           not_found := "ValidationSignals".FindPayload.not_found,
                           tail_address := "ValidationSignals".FindPayload.tail_address,
                           haystack := "LinkedList.IDB".list,
                           ENO => #_w1);
   IF #_w1 THEN "ValidationSignals".FindPayload.request := FALSE; END_IF;
END_REGION

REGION Network 4: VALIDATE FIND ID
   RUNG wire#powerrail
      Contact( "ValidationSignals".FindID.request )
      "LinkedList.FindID"(needle := "ValidationSignals".FindID.needle, not_found := "ValidationSignals".FindID.not_found, tail_address := "ValidationSignals".FindID.tail_address, haystack := "LinkedList.IDB".list, Ret_Val => "ValidationSignals".FindID.index)
      R_Coil( "ValidationSignals".FindID.request )
   END_RUNG
   // the same network as SCL:
   "ValidationSignals".FindID.index := "LinkedList.FindID"(EN := "ValidationSignals".FindID.request,
                           needle := "ValidationSignals".FindID.needle,
                           not_found := "ValidationSignals".FindID.not_found,
                           tail_address := "ValidationSignals".FindID.tail_address,
                           haystack := "LinkedList.IDB".list,
                           ENO => #_w1);
   IF #_w1 THEN "ValidationSignals".FindID.request := FALSE; END_IF;
END_REGION

REGION Network 5: VALIDATE FIND STATUS
   RUNG wire#powerrail
      Contact( "ValidationSignals".FindStatus.request )
      "LinkedList.FindStatus"(needle := "ValidationSignals".FindStatus.needle, not_found := "ValidationSignals".FindStatus.not_found, tail_address := "ValidationSignals".FindStatus.tail_address, haystack := "LinkedList.IDB".list, Ret_Val => "ValidationSignals".FindStatus.index)
      R_Coil( "ValidationSignals".FindStatus.request )
   END_RUNG
   // the same network as SCL:
   "ValidationSignals".FindStatus.index := "LinkedList.FindStatus"(EN := "ValidationSignals".FindStatus.request,
                           needle := "ValidationSignals".FindStatus.needle,
                           not_found := "ValidationSignals".FindStatus.not_found,
                           tail_address := "ValidationSignals".FindStatus.tail_address,
                           haystack := "LinkedList.IDB".list,
                           ENO => #_w1);
   IF #_w1 THEN "ValidationSignals".FindStatus.request := FALSE; END_IF;
END_REGION

REGION Network 6: VALIDATE ADD HEAD
   RUNG wire#powerrail
      Contact( "ValidationSignals".AddHead.request )
      "LinkedList.AddHead"(available_slot := "ValidationSignals".AddHead.available_slot, payload := "ValidationSignals".AddHead.payload, tail_address := "ValidationSignals".AddHead.tail_address, list := "LinkedList.IDB".list, Ret_Val => "ValidationSignals".AddHead.status)
      R_Coil( "ValidationSignals".AddHead.request )
   END_RUNG
   // the same network as SCL:
   "ValidationSignals".AddHead.status := "LinkedList.AddHead"(EN := "ValidationSignals".AddHead.request,
                           available_slot := "ValidationSignals".AddHead.available_slot,
                           payload := "ValidationSignals".AddHead.payload,
                           tail_address := "ValidationSignals".AddHead.tail_address,
                           list := "LinkedList.IDB".list,
                           ENO => #_w1);
   IF #_w1 THEN "ValidationSignals".AddHead.request := FALSE; END_IF;
END_REGION

REGION Network 7: VALIDATE REMOVE HEAD
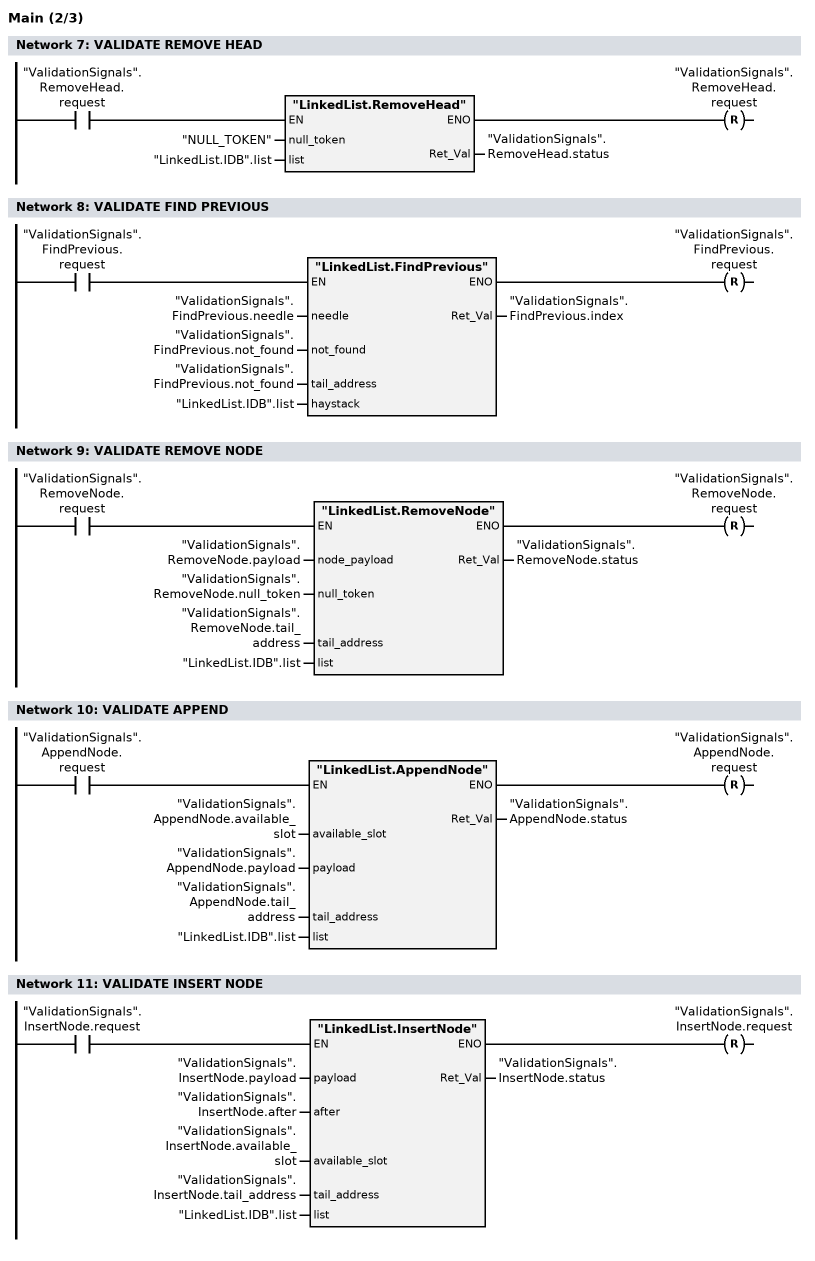
   RUNG wire#powerrail
      Contact( "ValidationSignals".RemoveHead.request )
      "LinkedList.RemoveHead"(null_token := "NULL_TOKEN", list := "LinkedList.IDB".list, Ret_Val => "ValidationSignals".RemoveHead.status)
      R_Coil( "ValidationSignals".RemoveHead.request )
   END_RUNG
   // the same network as SCL:
   "ValidationSignals".RemoveHead.status := "LinkedList.RemoveHead"(EN := "ValidationSignals".RemoveHead.request,
                           null_token := "NULL_TOKEN",
                           list := "LinkedList.IDB".list,
                           ENO => #_w1);
   IF #_w1 THEN "ValidationSignals".RemoveHead.request := FALSE; END_IF;
END_REGION

REGION Network 8: VALIDATE FIND PREVIOUS
   RUNG wire#powerrail
      Contact( "ValidationSignals".FindPrevious.request )
      "LinkedList.FindPrevious"(needle := "ValidationSignals".FindPrevious.needle, not_found := "ValidationSignals".FindPrevious.not_found, tail_address := "ValidationSignals".FindPrevious.not_found, haystack := "LinkedList.IDB".list, Ret_Val => "ValidationSignals".FindPrevious.index)
      R_Coil( "ValidationSignals".FindPrevious.request )
   END_RUNG
   // the same network as SCL:
   "ValidationSignals".FindPrevious.index := "LinkedList.FindPrevious"(EN := "ValidationSignals".FindPrevious.request,
                           needle := "ValidationSignals".FindPrevious.needle,
                           not_found := "ValidationSignals".FindPrevious.not_found,
                           tail_address := "ValidationSignals".FindPrevious.not_found,
                           haystack := "LinkedList.IDB".list,
                           ENO => #_w1);
   IF #_w1 THEN "ValidationSignals".FindPrevious.request := FALSE; END_IF;
END_REGION

REGION Network 9: VALIDATE REMOVE NODE
   RUNG wire#powerrail
      Contact( "ValidationSignals".RemoveNode.request )
      "LinkedList.RemoveNode"(node_payload := "ValidationSignals".RemoveNode.payload, null_token := "ValidationSignals".RemoveNode.null_token, tail_address := "ValidationSignals".RemoveNode.tail_address, list := "LinkedList.IDB".list, Ret_Val => "ValidationSignals".RemoveNode.status)
      R_Coil( "ValidationSignals".RemoveNode.request )
   END_RUNG
   // the same network as SCL:
   "ValidationSignals".RemoveNode.status := "LinkedList.RemoveNode"(EN := "ValidationSignals".RemoveNode.request,
                           node_payload := "ValidationSignals".RemoveNode.payload,
                           null_token := "ValidationSignals".RemoveNode.null_token,
                           tail_address := "ValidationSignals".RemoveNode.tail_address,
                           list := "LinkedList.IDB".list,
                           ENO => #_w1);
   IF #_w1 THEN "ValidationSignals".RemoveNode.request := FALSE; END_IF;
END_REGION

REGION Network 10: VALIDATE APPEND
   RUNG wire#powerrail
      Contact( "ValidationSignals".AppendNode.request )
      "LinkedList.AppendNode"(available_slot := "ValidationSignals".AppendNode.available_slot, payload := "ValidationSignals".AppendNode.payload, tail_address := "ValidationSignals".AppendNode.tail_address, list := "LinkedList.IDB".list, Ret_Val => "ValidationSignals".AppendNode.status)
      R_Coil( "ValidationSignals".AppendNode.request )
   END_RUNG
   // the same network as SCL:
   "ValidationSignals".AppendNode.status := "LinkedList.AppendNode"(EN := "ValidationSignals".AppendNode.request,
                           available_slot := "ValidationSignals".AppendNode.available_slot,
                           payload := "ValidationSignals".AppendNode.payload,
                           tail_address := "ValidationSignals".AppendNode.tail_address,
                           list := "LinkedList.IDB".list,
                           ENO => #_w1);
   IF #_w1 THEN "ValidationSignals".AppendNode.request := FALSE; END_IF;
END_REGION

REGION Network 11: VALIDATE INSERT NODE
   RUNG wire#powerrail
      Contact( "ValidationSignals".InsertNode.request )
      "LinkedList.InsertNode"(payload := "ValidationSignals".InsertNode.payload, after := "ValidationSignals".InsertNode.after, available_slot := "ValidationSignals".InsertNode.available_slot, tail_address := "ValidationSignals".InsertNode.tail_address, list := "LinkedList.IDB".list, Ret_Val => "ValidationSignals".InsertNode.status)
      R_Coil( "ValidationSignals".InsertNode.request )
   END_RUNG
   // the same network as SCL:
   "ValidationSignals".InsertNode.status := "LinkedList.InsertNode"(EN := "ValidationSignals".InsertNode.request,
                           payload := "ValidationSignals".InsertNode.payload,
                           after := "ValidationSignals".InsertNode.after,
                           available_slot := "ValidationSignals".InsertNode.available_slot,
                           tail_address := "ValidationSignals".InsertNode.tail_address,
                           list := "LinkedList.IDB".list,
                           ENO => #_w1);
   IF #_w1 THEN "ValidationSignals".InsertNode.request := FALSE; END_IF;
END_REGION

REGION Network 12: VALIDATE CLEAR LIST
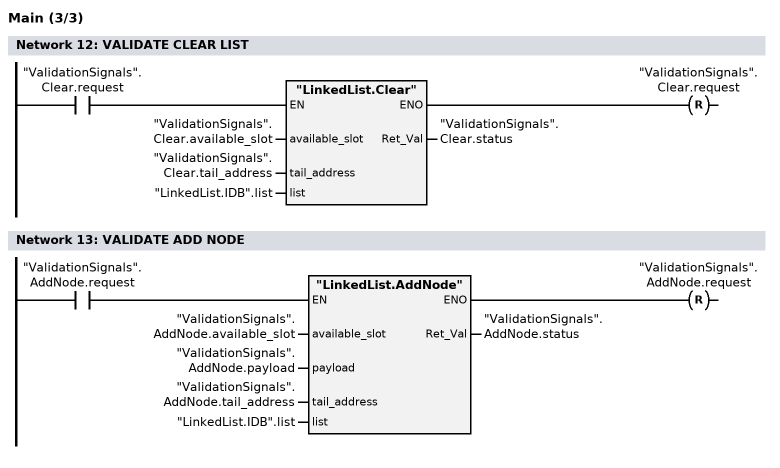
   RUNG wire#powerrail
      Contact( "ValidationSignals".Clear.request )
      "LinkedList.Clear"(available_slot := "ValidationSignals".Clear.available_slot, tail_address := "ValidationSignals".Clear.tail_address, list := "LinkedList.IDB".list, Ret_Val => "ValidationSignals".Clear.status)
      R_Coil( "ValidationSignals".Clear.request )
   END_RUNG
   // the same network as SCL:
   "ValidationSignals".Clear.status := "LinkedList.Clear"(EN := "ValidationSignals".Clear.request,
                           available_slot := "ValidationSignals".Clear.available_slot,
                           tail_address := "ValidationSignals".Clear.tail_address,
                           list := "LinkedList.IDB".list,
                           ENO => #_w1);
   IF #_w1 THEN "ValidationSignals".Clear.request := FALSE; END_IF;
END_REGION

REGION Network 13: VALIDATE ADD NODE
   RUNG wire#powerrail
      Contact( "ValidationSignals".AddNode.request )
      "LinkedList.AddNode"(available_slot := "ValidationSignals".AddNode.available_slot, payload := "ValidationSignals".AddNode.payload, tail_address := "ValidationSignals".AddNode.tail_address, list := "LinkedList.IDB".list, Ret_Val => "ValidationSignals".AddNode.status)
      R_Coil( "ValidationSignals".AddNode.request )
   END_RUNG
   // the same network as SCL:
   "ValidationSignals".AddNode.status := "LinkedList.AddNode"(EN := "ValidationSignals".AddNode.request,
                           available_slot := "ValidationSignals".AddNode.available_slot,
                           payload := "ValidationSignals".AddNode.payload,
                           tail_address := "ValidationSignals".AddNode.tail_address,
                           list := "LinkedList.IDB".list,
                           ENO => #_w1);
   IF #_w1 THEN "ValidationSignals".AddNode.request := FALSE; END_IF;
END_REGION
END_ORGANIZATION_BLOCK